// TwinCAT 3 PLC project DistanceSensor
// ProgramVersion: 3.1.4023.0
// libraries:
//   Tc2_SerialCom, * (Beckhoff Automation GmbH)
//   Tc2_Standard, * (Beckhoff Automation GmbH)
//   Tc2_System, * (Beckhoff Automation GmbH)
//   Tc3_Module, * (Beckhoff Automation GmbH)
// project tree:
//   DistanceSensor/ DistanceSensor.TcGVL, FB_DistanceSensor.TcPOU, FB_SerialComRS422.TcPOU
//   Outdated/ A_README.TcGVL, ILD1420.TcPOU, GVL_SerialBuffers.TcGVL (not stored), SerialComms_EL6021_ILD1420.TcPOU (not stored)
//   / PlcTask.TcTTO
//   POUs/ MAIN.TcPOU
// real-time tasks:
//   TASK PlcTask: cycle T#1ms, priority 20, ADS port 350
// I/O:
//   DEVICE Gerät 1 (EtherCAT), AmsNetId 10.183.66.136.2.1
//     Klemme 1 (EK1100) [EK1100 EtherCAT-Koppler (2A E-Bus)]
//       Klemme 2 (EL6021) [EL6021 Schnittstelle (RS422/485)]
//       Klemme 3 (EL6001) [EL6001 Schnittstelle (RS232)]
//       Klemme 4 (EL6001) [EL6001 Schnittstelle (RS232)]
//       Klemme 5 (EL2564) [EL2564 4 K. LED-Ausgang, 5...48 V DC, 4 A, RGBW]
//       Klemme 6 (EL9011) [EL9011 Endklemme]
// variable links:
//   DistanceSensor/DistanceSensor Instance <-> Device 1 (EtherCAT)/Term 1 (EK1100)/Term 2 (EL6021)
//     PlcTask Inputs/DistanceSensor.stEL6021In @bit {16..184 step 8} <-> COM TxPDO-Map Inputs/Data In {0..21}  (22 links)
//     PlcTask Inputs/DistanceSensor.stEL6021In <-> COM TxPDO-Map Inputs/Status
//     PlcTask Outputs/DistanceSensor.stEL6021Out <-> COM RxPDO-Map Outputs/Ctrl
//     PlcTask Outputs/DistanceSensor.stEL6021Out @bit {16..184 step 8} <-> COM RxPDO-Map Outputs/Data Out {0..21}  (22 links)

CONFIGURATION DistanceSensor
    RESOURCE PLC ON TwinCAT3
        TASK PlcTask(INTERVAL := T#1ms, PRIORITY := 20);
        PROGRAM MAIN WITH PlcTask : MAIN;
    END_RESOURCE
END_CONFIGURATION

// ---- DistanceSensor/DistanceSensor.TcGVL
{attribute 'qualified_only'}
VAR_GLOBAL
	stEL6021In  AT %I*	: EL6inData22B;		//**To EL6021 Inputs**
	stEL6021Out AT %Q*	: EL6outData22B;	//**To EL6021 Outputs**
END_VAR

// How to use ILD1420 Distance Sensor (digital Output) with El6021 clamp:
//
// 1. Add 'Tc2_SerialCom' to references 
// 2. Map EL6021 Inputs (including status) with stEL6021In in GVL DistanceSensor
// 3. Map EL6021 Outputs (including ctrl) with stEL6021Out in GVL DistanceSensor
// 4. Call FB_DistanceSensor in MAIN
// 5. Make sure Task cycle time is small enough (recommended 1 ms)
// 6. Make sure Baud rates of Sensor and Clamp align (115200) (CoE Online Settings)
// 7. Outdated folder contains original version with background program

// ---- Outdated/A_README.TcGVL
VAR_GLOBAL
	// How to use ILD1420 Distance Sensor (digital Output) with El6021 clamp:
	//
	// 1. Add 'Tc2_SerialCom' to references
	// 2. change 'dNumOfSensors' in 'GVL_SerialBuffers' to the amount of senors connected to a Beckhoff coupler or PLC
	//		-> all variables and %I*/%Q* are automaticly adjusted to the amount of desired ILD1420 sensors
	// 3. PRG SerialComms_EL6021_ILD1420() needs to be called in MAIN 
	// 4. Objects of FB ILD1420 can now be initialized according to it's input variables 
	//		(example: ILD1420_Sensor1(RxBuffer := GVL_SerialBuffers.RxBufferEL[0]);		// init sensor 1
	//				  ILD1420_Sensor2(RxBuffer := GVL_SerialBuffers.RxBufferEL[1]);		// init sensor 2)
	// 5. Connect 'COM TxPDO-Map Inputs' and 'COM RxPDO-Map Outputs' to PLC variables
	//		HINT: Code needs be be build once in order for PLC to find all In-/Output variables
	//		HINT: ALL Inputs and Outputs (Status, Data In [0..21], Ctrl & Data Out [0..21] need to be connected, even if Tx is not needed
END_VAR

// ---- POUs/MAIN.TcPOU
PROGRAM MAIN
VAR
	fbDistanceSensor : FB_DistanceSensor;
	
	fDistance : LREAL;
END_VAR

fbDistanceSensor();
fDistance := fbDistanceSensor.fDistance;

END_PROGRAM

// ---- DistanceSensor/FB_DistanceSensor.TcPOU
FUNCTION_BLOCK FB_DistanceSensor
VAR_OUTPUT
	fDistance 			: LREAL;
END_VAR
VAR
	//Local
	fbEL6021			: FB_SerialComRS422;

	//ErrorBits
	bCommunicationError : BIT;
	bOutOfRange 		: BIT;
END_VAR
VAR CONSTANT
	fSMR 		: LREAL := 50.0;				// Start of Measuring Range
	fEMR 		: LREAL := 150.0;				// End of Measuring Range
END_VAR

fbEL6021(stReceiveData:=DistanceSensor.stEL6021In, stTransmitData:=DistanceSensor.stEL6021Out);

fDistance := fbEL6021.fDistance;

END_FUNCTION_BLOCK

// ---- DistanceSensor/FB_SerialComRS422.TcPOU
FUNCTION_BLOCK FB_SerialComRS422
VAR_IN_OUT
	stReceiveData 	: EL6inData22B;
	stTransmitData 	: EL6outData22B;
END_VAR
VAR_OUTPUT
	fDistance : LREAL;
	eReceiveErrorID	: ComError_t;
END_VAR
VAR
	//Receive Buffer
	fbEL6021Ctrl					: SerialLineControl;
	RxBuffer 						: ComBuffer;
	TxBuffer						: ComBuffer;
	//Receive Data
	fbReceiveByte					: ReceiveByte;				
	nFirstThreeBytesOfBuffer  		: ARRAY[0..2] OF BYTE;		// buffer storage for the three bytes that contain the distance information
	nRcvIndex						: UINT := 0;				// Counter
	nDistanceAsStringOfBits			: DINT;
END_VAR
VAR CONSTANT
	fSMR 		: LREAL := 50.0;				// Start of Measuring Range
	fEMR 		: LREAL := 150.0;				// End of Measuring Range
END_VAR

fbEL6021Ctrl(
			Mode:= SERIALLINEMODE_EL6_22B,
			pComIn:= ADR(stReceiveData),
			pComOut:= ADR(stTransmitData),
			SizeComIn:= SIZEOF(stReceiveData),
			Error=>,
			ErrorID=>,
			TxBuffer:=TxBuffer,
			RxBuffer:=RxBuffer,);

fbReceiveByte(RXbuffer := RxBuffer, Error => eReceiveErrorID);

WHILE fbReceiveByte.ByteReceived AND (nRcvIndex <= SIZEOF(nFirstThreeBytesOfBuffer)) DO
	fbReceiveByte(RXbuffer := RxBuffer);
	IF (fbReceiveByte.ReceivedByte.7) = 0 THEN
		nFirstThreeBytesOfBuffer[nRcvIndex] := fbReceiveByte.ReceivedByte;
		nRcvIndex := nRcvIndex + 1;
	ELSE
		nFirstThreeBytesOfBuffer[2] := fbReceiveByte.ReceivedByte;
		nRcvIndex	:= 0;
	END_IF
END_WHILE

doSortBits(nByteBuffer:=nFirstThreeBytesOfBuffer);
doConvertToDistanceValue(nBitString:=nDistanceAsStringOfBits, fMax:=fEMR, fMin:=fSMR);

METHOD PRIVATE doConvertToDistanceValue
VAR_INPUT
	nBitString : DINT;
	fMax : LREAL;
	fMIn : LREAL;
END_VAR
fDistance := 50.0 + 1.0/100.0 * (102.0/65520.0 * DINT_TO_LREAL(nBitString) - 1.0) * (fMax - fMIn);
END_METHOD

METHOD PRIVATE doSortBits
VAR_INPUT
	nByteBuffer : ARRAY [0..2] OF BYTE;
END_VAR
// Rearrange L,M,H Refer Pg 85. We seperate the distance bits from the error, transmissions, ect. -bits in this step.
// MemCopy is a possilbe way to simplify code. But since we need to work with bit and not buyts, this is actually the more readable code.
// Also TwinCAT demands CONST values when working with bit handeling, so loops are also not possible.
nDistanceAsStringOfBits.0 	:= nByteBuffer[0].0;
nDistanceAsStringOfBits.1 	:= nByteBuffer[0].1;
nDistanceAsStringOfBits.2 	:= nByteBuffer[0].2;
nDistanceAsStringOfBits.3 	:= nByteBuffer[0].3;
nDistanceAsStringOfBits.4 	:= nByteBuffer[0].4;
nDistanceAsStringOfBits.5 	:= nByteBuffer[0].5;
nDistanceAsStringOfBits.6 	:= nByteBuffer[1].0;
nDistanceAsStringOfBits.7 	:= nByteBuffer[1].1;
nDistanceAsStringOfBits.8 	:= nByteBuffer[1].2;
nDistanceAsStringOfBits.9 	:= nByteBuffer[1].3;
nDistanceAsStringOfBits.10 	:= nByteBuffer[1].4;
nDistanceAsStringOfBits.11	:= nByteBuffer[1].5;
nDistanceAsStringOfBits.12 	:= nByteBuffer[2].0;
nDistanceAsStringOfBits.13 	:= nByteBuffer[2].1;
nDistanceAsStringOfBits.14 	:= nByteBuffer[2].2;
nDistanceAsStringOfBits.15 	:= nByteBuffer[2].3;
END_METHOD

END_FUNCTION_BLOCK

// ---- Outdated/ILD1420.TcPOU
// By Devika Ajith, Daniel Lindner and Oliver Schubert.
// June 2022
//
// This functionblock contains the logic needed to get a distance value from the raw RS422 bytes recieved BY an EL6021 clamp.
//

FUNCTION_BLOCK ILD1420
VAR_INPUT
	RxBuffer : ComBuffer;			// RxBuffer is used to pass data recieved by the EL6021 clap.
									// We expect the first 3 bytes of that buffer to contain data relevant to the distance measurement.
	
	//TxBuffer	: ComBuffer;		//Since the functionality provided BY THIS functionblock does NOT include ANY sending logic,
									//the TxBuffer is commented out FOR now. THIS might change with future functionality extensions.
END_VAR
VAR_OUTPUT
	lrDistance  : LREAL := 0;
	bInRange 	: BOOL;
END_VAR
VAR CONSTANT
	lrSMR 		: LREAL := 50.0;				// Start of Measuring Range
	lrEMR 		: LREAL := 150.0;				// End of Measuring Range
	lrMR  		: LREAL := lrEMR - lrSMR;		// Measuring Range
END_VAR
VAR
	//Receive data
	fbReceiveByte					: ReceiveByte;				
	first_three_bytes_of_rx_buffer  : ARRAY[0..2] OF BYTE;		// buffer storage for the three bytes that contain the distance information
	uiRcvIndex						: UINT := 0;				// Counter

	//decoding values
	diDistance_As_String_Of_Bits	: DINT;
END_VAR

// https://www.micro-epsilon.de/download/manuals/man--optoNCDT-1420--en.pdf
// Refer Pg 15 Resolution details
// Pg 84 - Byte decoding


fbReceiveByte(RXbuffer := RxBuffer);		// init FB fbReceiveByte with Buffer

// get received Bytes from the EL6021 and store them into an array of Bytes
// These bytes contain error, transmissions, ect. -bits and also the bits for the distance information.
// We store all bits and seperate the distance bits from the error, transmissions, ect. -bits in the next step
WHILE fbReceiveByte.ByteReceived AND (uiRcvIndex <= SIZEOF(first_three_bytes_of_rx_buffer)) DO
	fbReceiveByte(RXbuffer := RxBuffer);
	IF (fbReceiveByte.ReceivedByte.7) = 0 THEN
		first_three_bytes_of_rx_buffer[uiRcvIndex] := fbReceiveByte.ReceivedByte;
		uiRcvIndex := uiRcvIndex + 1;
	ELSE
		first_three_bytes_of_rx_buffer[2] := fbReceiveByte.ReceivedByte;
		uiRcvIndex	:= 0;
	END_IF
END_WHILE


// Rearrange L,M,H Refer Pg 85. We seperate the distance bits from the error, transmissions, ect. -bits in this step.
// MemCopy is a possilbe way to simplify code. But since we need to work with bit and not buyts, this is actually the more readable code.
// Also TwinCAT demands CONST values when working with bit handeling, so loops are also not possible.
diDistance_As_String_Of_Bits.0 	:= first_three_bytes_of_rx_buffer[0].0;
diDistance_As_String_Of_Bits.1 	:= first_three_bytes_of_rx_buffer[0].1;
diDistance_As_String_Of_Bits.2 	:= first_three_bytes_of_rx_buffer[0].2;
diDistance_As_String_Of_Bits.3 	:= first_three_bytes_of_rx_buffer[0].3;
diDistance_As_String_Of_Bits.4 	:= first_three_bytes_of_rx_buffer[0].4;
diDistance_As_String_Of_Bits.5 	:= first_three_bytes_of_rx_buffer[0].5;
diDistance_As_String_Of_Bits.6 	:= first_three_bytes_of_rx_buffer[1].0;
diDistance_As_String_Of_Bits.7 	:= first_three_bytes_of_rx_buffer[1].1;
diDistance_As_String_Of_Bits.8 	:= first_three_bytes_of_rx_buffer[1].2;
diDistance_As_String_Of_Bits.9 	:= first_three_bytes_of_rx_buffer[1].3;
diDistance_As_String_Of_Bits.10 := first_three_bytes_of_rx_buffer[1].4;
diDistance_As_String_Of_Bits.11	:= first_three_bytes_of_rx_buffer[1].5;
diDistance_As_String_Of_Bits.12 := first_three_bytes_of_rx_buffer[2].0;
diDistance_As_String_Of_Bits.13 := first_three_bytes_of_rx_buffer[2].1;
diDistance_As_String_Of_Bits.14 := first_three_bytes_of_rx_buffer[2].2;
diDistance_As_String_Of_Bits.15 := first_three_bytes_of_rx_buffer[2].3;


// conversion von bits to LREAL via formula from
// https://www.micro-epsilon.de/download/manuals/man--optoNCDT-1420--en.pdf
lrDistance := 50.0 + 1.0/100.0 * (102.0/65520.0 * DINT_TO_LREAL(diDistance_As_String_Of_Bits) - 1.0) * lrMR;

// to distinguish values wich are out of range, choose arbitrary value far away from SMR and EMR
IF lrDistance < lrSMR OR lrDistance > lrEMR THEN
	bInRange := FALSE;
	lrDistance := 999;
ELSE
	bInRange := TRUE;
END_IF

END_FUNCTION_BLOCK
